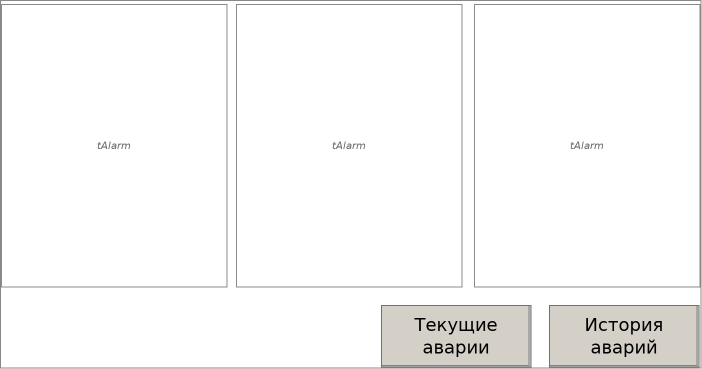
VISUALIZATION AlarmsVisSample  // 702x369
    Frame (1,4 226x283)
        shows tAlarm(alarm := Alarms.SeriosAlarm)
    Frame (236,4 226x283)
        shows tAlarm(alarm := Alarms.NotSeriosAlarm)
    Frame (474,4 226x283)
        shows tAlarm(alarm := Alarms.SimpleWarning)
    Button (381,305 150x62), "Текущие аварии"
        OnMouseClick: OpenDialog Dialog=Tc3_BAR_Common.Current_Alarms_dialog, OpenModal=True, OpenCentered=True
    Button (549,305 150x62), "История аварий"
        OnMouseClick: OpenDialog Dialog=Tc3_BAR_Common.History_Of_Alarms_dialog, OpenModal=True, OpenCentered=True
END_VISUALIZATION

(* stored: Version 1.1.0.1, ProductVersion 3.1.4024.2
   Visu AlarmsVisSample: Id {eb7f244c-7d80-454f-8411-c92c2d0b1de4} *)
